// TwinCAT 3 PLC project NitroLogger
// Title: Tc_EventLogger
// Company: Reinova s.p.a.
// Author: Lorenzo Musco
// ProjectVersion: 1.1.2.6
// Description: This library wrap a Function block around the pre-existing TcLog in order to avoid cyclic call to the logger.
// ProgramVersion: 3.1.4024.0
// libraries:
//   Tc2_Standard, * (Beckhoff Automation GmbH)
//   Tc2_System, * (Beckhoff Automation GmbH)
//   Tc2_Utilities, * (Beckhoff Automation GmbH)
//   Tc3_Module, * (Beckhoff Automation GmbH)
//   TcLog, * (Benedikt Geisler)
//   Base Interfaces,newest,System
//   Tc3_DynamicMemory,1.0.2.0,Beckhoff Automation GmbH
// project tree:
//   / PlcTask.TcTTO
//   POUs/FB/ FB_EventLogger.TcPOU, FB_EventLoggerCore.TcPOU, FB_LogTrig.TcPOU, LogLevelToAdsLogMsgType.TcPOU
//   POUs/StringBuilder/ StringBuilder.TcPOU
//   POUs/StringBuilder/_Interfaces/ ILimitedStringBuilder.TcIO, IStringBuilder.TcIO
//   POUs/Utils/ AnyToString.TcPOU, DateTime.TcPOU, DeleteOldFiles.TcPOU, DynamicStringBuffer.TcPOU, GetFileAgeInSeconds.TcPOU
//   POUs/Utils/_DataTypes/ DeleteFilesState.TcDUT, PersistToFileState.TcDUT
//   POUs/_DataTypes/ Error.TcDUT, ErrorCodes.TcDUT, LoggingConfiguration.TcDUT, LogLevels.TcDUT, RollingIntervals.TcDUT
//   Version/ Global_Version.TcGVL
// real-time tasks:
//   TASK PlcTask: cycle T#10ms, priority 20, ADS port 350

CONFIGURATION NitroLogger
    RESOURCE PLC ON TwinCAT3
        TASK PlcTask(INTERVAL := T#10ms, PRIORITY := 20);
        PROGRAM MAIN WITH PlcTask : MAIN;
    END_RESOURCE
END_CONFIGURATION

// ---- POUs/Utils/_DataTypes/DeleteFilesState.TcDUT
// States for state machine used in `DeleteOldFiles`.
{attribute 'qualified_only'}
{attribute 'strict'}
TYPE INTERNAL DeleteFilesState :
(
	Idle := 0,
  SearchNextFile,
  WaitUntilExecutionDone,
  ProcessFoundFiles,
  CheckIfFileIsDirectory,
  CheckFileTime,
  DeleteFile,
  FileDeleted
);
END_TYPE

// ---- POUs/Utils/_DataTypes/PersistToFileState.TcDUT
// States for state machine used in `DynamicStringBuffer.PersistToFile`
{attribute 'qualified_only'}
{attribute 'strict'}
TYPE INTERNAL PersistToFileState :
(
	Idle := 0,
  OpenFile,
  GetStringFromFifo,
  AppendDataToFile,
  CloseFile
);
END_TYPE

// ---- POUs/_DataTypes/Error.TcDUT
/// This is the error type used in this library.
TYPE Error :
STRUCT
  /// `TRUE` signals an active error
	Active : BOOL;
  /// Error code of type `ErrorCodes`
	Code : INT;
  /// Plain text error message
	Info : Tc2_System.T_MaxString;
END_STRUCT
END_TYPE

// ---- POUs/_DataTypes/ErrorCodes.TcDUT
/// Provides error codes for TcLogCore
{attribute 'qualified_only'}
{attribute 'strict'}
{attribute 'to_string'}
TYPE ErrorCodes : 
(
	None := 0,
	OpeningFileFailed,
	WritingToFileFailed,
	ClosingFileFailed,
	EnumeratingFilesInSpecifiedDirectoryFailed,
	DeletingFileFailed,
	FifoOverflow
);
END_TYPE

// ---- POUs/_DataTypes/LoggingConfiguration.TcDUT
/// Configuration of TcLogCore
TYPE LoggingConfiguration :
STRUCT
  /// File name where the logs should be written to. Should not include path.
	FileName : Tc2_System.T_MaxString;
  /// File path where the logs should be written to. Will be prefixed to `FileName`
	FilePath : Tc2_System.T_MaxString;
  /// Whether to include the instance path of TcLog into the log message or not.
	IncludeInstancePath : BOOL;
  /// Whether to write the logs to ADS output or not.
	WriteToAds : BOOL;
  /// Rolling interval: when to create a new log file.
	RollingInterval : RollingIntervals;
  /// What is the minimum log level that gets logged?
	MinimumLevel : LogLevels;
  /// Which delimiter should be used between the different parts of the log string?
	Delimiter : STRING(1);
  /// When should old log files be deleted? Unit: days. Set it to `0` if log files should never be deleted. 
	LogFileLifespan : UINT;
  /// Format of timestamp. See `TcLogCore.TimestampFormat` for formatting options.
	TimestampFormat : STRING;
END_STRUCT
END_TYPE

// ---- POUs/_DataTypes/LogLevels.TcDUT
/// Log level of message to be logged.
{attribute 'qualified_only'}
{attribute 'strict'}
{attribute 'to_string'}
TYPE LogLevels :
(
	Debug := 0,
	Information,
	Warning,
	Error,
	Fatal
);
END_TYPE

// ---- POUs/_DataTypes/RollingIntervals.TcDUT
/// Rolling interval to create a new log file when expired. 
{attribute 'qualified_only'}
{attribute 'strict'}
{attrivute 'to_string'}
TYPE RollingIntervals :
(
	None := 0,
	Hourly,
	Daily,
	Monthly
);
END_TYPE

// ---- Version/Global_Version.TcGVL
{attribute 'TcGenerated'}
{attribute 'no-analysis'}
{attribute 'linkalways'}
// This function has been automatically generated from the project information.
VAR_GLOBAL CONSTANT
	{attribute 'const_non_replaced'}
	stLibVersion_Tc_EventLogger : ST_LibVersion := (iMajor := 1, iMinor := 1, iBuild := 2, iRevision := 6, nFlags := 1, sVersion := '1.1.2.6');
END_VAR

// ---- POUs/StringBuilder/_Interfaces/ILimitedStringBuilder.TcIO
{attribute 'hide'}
INTERFACE INTERNAL ILimitedStringBuilder

METHOD Append : IStringBuilder // Append text TO t current build STRING.
VAR_INPUT
    Text : Tc2_System.T_MaxString; //Text to append to current build string
END_VAR
END_METHOD

METHOD AppendIf : IStringBuilder
VAR_INPUT
    Condition : BOOL;
    Text : Tc2_System.T_MaxString;
END_VAR
END_METHOD

METHOD Reset : ILimitedStringBuilder //Reset current build STRING TO an empty STRING.
END_METHOD

METHOD ToString : Tc2_System.T_MaxString //Returns current build STRING.
END_METHOD

END_INTERFACE

// ---- POUs/StringBuilder/_Interfaces/IStringBuilder.TcIO
{attribute 'hide'}
INTERFACE INTERNAL IStringBuilder

METHOD Append : IStringBuilder // Append text TO t current build STRING.
VAR_INPUT
    Text : Tc2_System.T_MaxString; //Text to append to current build string
END_VAR
END_METHOD

METHOD AppendIf : IStringBuilder
VAR_INPUT
    Condition : BOOL;
    Text : Tc2_System.T_MaxString;
END_VAR
END_METHOD

METHOD InsertAtLocation : IStringBuilder
VAR_INPUT
    Text : Tc2_System.T_MaxString;
    Position : INT;
END_VAR
END_METHOD

METHOD PadLeft : IStringBuilder
VAR_INPUT
    Text : Tc2_System.T_MaxString; // Text to append to current build string
    Length : INT; // Total length of text + padding
    Char : STRING(1); // Character to be padded left of text
END_VAR
END_METHOD

METHOD Reset : ILimitedStringBuilder //Reset current build STRING TO an empty STRING.
END_METHOD

METHOD ToString : Tc2_System.T_MaxString //Returns current build STRING.
END_METHOD

END_INTERFACE

// ---- POUs/FB/FB_EventLogger.TcPOU
{attribute 'reflection'} 
FUNCTION_BLOCK FB_EventLogger EXTENDS TcLog
VAR
	_WorkString			: Tc2_System.T_MaxString;
	isSpammable			: BOOL;
	
	OldsCompletedString, NewCompletedString : T_MaxString;
END_VAR

METHOD Append : REFERENCE TO FB_EventLogger
VAR_INPUT
	sString		: T_MaxString;
END_VAR

VAR_INST
	OldString 	: T_MaxString;
END_VAR
_WorkString := CONCAT(_WorkString, sString);

Append REF= THIS^;
END_METHOD

METHOD CanSpam : REFERENCE TO FB_EventLogger
VAR
	
END_VAR
isSpammable := TRUE; 
CanSpam REF= THIS^;
END_METHOD

/// Logs the log string in DEBUG level.
METHOD Debug : BOOL
VAR_INPUT
  	message : T_MaxString; 
END_VAR
_WorkString := CONCAT(_WorkString, message);
NewCompletedString := _WorkString;
_WorkString := '';

IF NewCompletedString <> OldsCompletedString OR isSpammable THEN
	SUPER^.Debug(NewCompletedString);
	OldsCompletedString := NewCompletedString;
	isSpammable := FALSE;
END_IF
END_METHOD

/// Logs the log string in ERROR level.
METHOD Error : BOOL
VAR_INPUT
  	message : T_MaxString; 
END_VAR
_WorkString := CONCAT(_WorkString, message);
NewCompletedString := _WorkString;
_WorkString := '';

IF NewCompletedString <> OldsCompletedString THEN
	SUPER^.Error(NewCompletedString);
	OldsCompletedString := NewCompletedString;
	isSpammable := FALSE;
END_IF
END_METHOD

/// Logs the log string in FATAL level.
METHOD Fatal : BOOL
VAR_INPUT
  	message : T_MaxString; 
END_VAR
_WorkString := CONCAT(_WorkString, message);
NewCompletedString := _WorkString;
_WorkString := '';

IF NewCompletedString <> OldsCompletedString THEN
	SUPER^.Error(NewCompletedString);
	OldsCompletedString := NewCompletedString;
	isSpammable := FALSE;
END_IF
END_METHOD

/// Logs the log string in INFORMATION level.
METHOD Information : BOOL
VAR_INPUT
  	message : T_MaxString; 
END_VAR
_WorkString := CONCAT(_WorkString, message);
NewCompletedString := _WorkString;
_WorkString := '';

IF NewCompletedString <> OldsCompletedString THEN
	SUPER^.Information(NewCompletedString);
	OldsCompletedString := NewCompletedString;
	isSpammable := FALSE;
END_IF
END_METHOD

/// Initializes the reference to the core logger. Should only be called once from the core logger directly.
METHOD PUBLIC Init : BOOL
VAR_INPUT
  /// Reference to TcLoggerCore instance.
  ref2Core : ILogCore; 
END_VAR
SUPER^.Init(ref2Core);
END_METHOD

/// Logs the log string in WARNING level.
METHOD Warning : BOOL
VAR_INPUT
  	message : T_MaxString; 
END_VAR
_WorkString := CONCAT(_WorkString, message);
NewCompletedString := _WorkString;
_WorkString := '';

IF NewCompletedString <> OldsCompletedString THEN
	SUPER^.Warning(NewCompletedString);
	OldsCompletedString := NewCompletedString;
	isSpammable := FALSE;
END_IF
END_METHOD

END_FUNCTION_BLOCK

// ---- POUs/FB/FB_EventLoggerCore.TcPOU
FUNCTION_BLOCK FB_EventLoggerCore EXTENDS TcLogCore
VAR_INPUT
END_VAR
VAR_OUTPUT
END_VAR
VAR
END_VAR

END_FUNCTION_BLOCK

// ---- POUs/FB/FB_LogTrig.TcPOU
/// This function block can be used to log on rising or falling edges.
/// For each signal that should be watched, a separate instance of `TcLogTrig` 
/// must be created.
FUNCTION_BLOCK FB_LogTrig EXTENDS TcLog

/// Logs data on falling edge of `CLK`.
{attribute 'hide_all_locals'}
METHOD OnFallingEdge : REFERENCE TO TcLog
VAR_INPUT
  /// Falling edge triggers logging the data.
  CLK : BOOL; 
END_VAR
VAR_INST
    fTrig : Tc2_Standard.F_TRIG;
END_VAR
fTrig(CLK:=CLK);

SUPER^.OnCondition(fTrig.Q);

OnFallingEdge REF= THIS^;
END_METHOD

/// Logs data on rising edge of `CLK`.
{attribute 'hide_all_locals'}
METHOD OnRisingEdge : REFERENCE TO TcLog
VAR_INPUT
  /// Rising edge logs data.
  CLK : BOOL; 
END_VAR
VAR_INST
    rTrig : Tc2_Standard.R_TRIG;
END_VAR
rTrig(CLK:=CLK);

SUPER^.OnCondition(rTrig.Q);

OnRisingEdge REF= THIS^;
END_METHOD

END_FUNCTION_BLOCK

// ---- POUs/FB/LogLevelToAdsLogMsgType.TcPOU
// Converts TcLog.LogLevels into Tc2_System.ADSLOG_MSGTYPEs.
{attribute 'hide'}
FUNCTION INTERNAL LogLevelToAdsLogMsgType : DWORD
VAR_INPUT
  logLevel : LogLevels;
END_VAR
VAR
  _retVal : DWORD;
END_VAR

CASE logLevel OF
  LogLevels.Debug, LogLevels.Information:
    _retVal := Tc2_System.ADSLOG_MSGTYPE_HINT;
  LogLevels.Warning:
    _retVal := Tc2_System.ADSLOG_MSGTYPE_WARN;
  LogLevels.Error, LogLevels.Fatal:
    _retVal := Tc2_System.ADSLOG_MSGTYPE_ERROR;
  ELSE
    _retVal := Tc2_System.ADSLOG_MSGTYPE_HINT;
END_CASE

LogLevelToAdsLogMsgType := _retVal;

END_FUNCTION

// ---- POUs/StringBuilder/StringBuilder.TcPOU
FUNCTION_BLOCK INTERNAL StringBuilder IMPLEMENTS IStringBuilder, ILimitedStringBuilder
VAR
  {attribute 'hide'}
  _workString : Tc2_System.T_MaxString;
END_VAR

METHOD PUBLIC Append : IStringBuilder // Append text TO t current build STRING.
VAR_INPUT
  text : Tc2_System.T_MaxString; //text to append to current build string
END_VAR
_workString:= Tc2_Standard.CONCAT(_workString,text);
Append := THIS^;
END_METHOD

METHOD PUBLIC AppendIf : IStringBuilder
VAR_INPUT
  condition : BOOL;
  text : Tc2_System.T_MaxString;
END_VAR
IF condition THEN
  _workString:= Tc2_Standard.CONCAT(_workString,text);
END_IF
AppendIf := THIS^;
END_METHOD

METHOD PUBLIC InsertAtLocation : IStringBuilder
VAR_INPUT
  text : Tc2_System.T_MaxString;
  position : INT;
END_VAR
_workString := Tc2_Standard.INSERT(_workSTring,text,position);
InsertAtLocation  := THIS^;
END_METHOD

METHOD PadLeft : IStringBuilder
VAR_INPUT
  text : Tc2_System.T_MaxString; // Text to append to current build string
  length : INT; // Total length of text + padding
  char : STRING(1); // Character to be padded left of text
END_VAR
VAR
  i : INT;
  padLength : INT;
END_VAR
// Add left padding
padLength := Tc2_Standard.LEN(text) - length;
FOR i := 1 TO padLength DO
  _workString:= Tc2_Standard.CONCAT(_workString, char);
END_FOR

// Add text
_workString:= Tc2_Standard.CONCAT(_workString,text);

PadLeft := THIS^;
END_METHOD

METHOD PUBLIC Reset : ILimitedStringBuilder //Reset current build STRING TO an empty STRING.
_workString:='';
Reset := THIS^;
END_METHOD

METHOD PUBLIC ToString : Tc2_System.T_MaxString //Returns current build STRING.
ToString := _workString;
END_METHOD

END_FUNCTION_BLOCK

// ---- POUs/Utils/AnyToString.TcPOU
/// Converts value of input data to string, where the input type can be any of 
/// the standard data types.
FUNCTION AnyToString : Tc2_System.T_MaxString
VAR_INPUT
  /// Input data
  data : ANY;
END_VAR
VAR
  _anyByte : POINTER TO BYTE;
  _anyUSINT : POINTER TO USINT;
  _anyInt : POINTER TO INT;
  _anyUInt : POINTER TO UINT;
  _anyUDInt : POINTER TO UDINT;
  _anySInt : POINTER TO SINT;
  _anyDInt : POINTER TO DINT;
  _anyLInt : POINTER TO LINT;
  _anyULInt : POINTER TO ULINT;
  _anyWord : POINTER TO WORD;
  _anyLWord : POINTER TO LWORD;
  _anyReal : POINTER TO REAL;
  _anyLReal : POINTER TO LREAL;
  _anyDateAndTime : POINTER TO DATE_AND_TIME;
  _anyDate : POINTER TO DATE;
  _anyTime : POINTER TO TIME;
  _anyWString : POINTER TO WSTRING;
  _anyTOD : POINTER TO TOD;
  _anyString : POINTER TO STRING;
  _string : T_MAXSTRING;
  _wString : WSTRING;
END_VAR

IF data.TypeClass = __SYSTEM.TYPE_CLASS.TYPE_BYTE THEN
  _anyByte := data.pValue;
  AnyToString := BYTE_TO_STRING(_anyByte^);
    
ELSIF data.TypeClass = __SYSTEM.TYPE_CLASS.TYPE_INT THEN
  _anyInt := data.pValue;
  AnyToString := INT_TO_STRING(_anyInt^);
    
ELSIF data.TypeClass = __SYSTEM.TYPE_CLASS.TYPE_UINT THEN
  _anyUInt := data.pValue;
  AnyToString := UINT_TO_STRING(_anyUInt^);
    
ELSIF data.TypeClass = __SYSTEM.TYPE_CLASS.TYPE_UDINT THEN
  _anyUDInt := data.pValue;
  AnyToString := UDINT_TO_STRING(_anyUDInt^);
    
ELSIF data.TypeClass = __SYSTEM.TYPE_CLASS.TYPE_SINT THEN
  _anySInt := data.pValue;
  AnyToString := SINT_TO_STRING(_anySInt^);
    
ELSIF data.TypeClass = __SYSTEM.TYPE_CLASS.TYPE_USINT THEN
  _anyUSInt := data.pValue;
  AnyToString := USINT_TO_STRING(_anyUSInt^);
    
ELSIF data.TypeClass = __SYSTEM.TYPE_CLASS.TYPE_DINT THEN
  _anyDInt := data.pValue;
  AnyToString := DINT_TO_STRING(_anyDInt^);
    
ELSIF data.TypeClass = __SYSTEM.TYPE_CLASS.TYPE_LINT THEN
  _anyLInt := data.pValue;
  AnyToString := LINT_TO_STRING(_anyLInt^);
      
ELSIF data.TypeClass = __SYSTEM.TYPE_CLASS.TYPE_ULINT THEN
  _anyULInt := data.pValue;
  AnyToString := ULINT_TO_STRING(_anyULInt^);
  
ELSIF data.TypeClass = __SYSTEM.TYPE_CLASS.TYPE_WORD THEN
  _anyWord := data.pValue;
  AnyToString := WORD_TO_STRING(_anyWord^);
    
ELSIF data.TypeClass = __SYSTEM.TYPE_CLASS.TYPE_LWORD THEN
  _anyLWord := data.pValue;
  AnyToString := LWORD_TO_STRING(_anyLWord^);
  
ELSIF data.TypeClass = __SYSTEM.TYPE_CLASS.TYPE_REAL THEN
  _anyReal := data.pValue;
  AnyToString := REAL_TO_STRING(_anyReal^);
  
ELSIF data.TypeClass = __SYSTEM.TYPE_CLASS.TYPE_LREAL THEN
  _anyLReal := data.pValue;
  AnyToString := LREAL_TO_STRING(_anyLReal^);
  
ELSIF data.TypeClass = __SYSTEM.TYPE_CLASS.TYPE_DATEANDTIME THEN
  _anyDateAndTime := data.pValue;
  AnyToString := DT_TO_STRING(_anyDateAndTime^);  
  
ELSIF data.TypeClass = __SYSTEM.TYPE_CLASS.TYPE_DATE THEN
  _anyDate := data.pValue;
  AnyToString := DATE_TO_STRING(_anyDate^);
  
ELSIF data.TypeClass = __SYSTEM.TYPE_CLASS.TYPE_TIME THEN
  _anyTime := data.pValue;
  AnyToString := TIME_TO_STRING(_anyTime^);
  
ELSIF data.TypeClass = __SYSTEM.TYPE_CLASS.TYPE_STRING THEN
  _anyString := data.pValue;
  AnyToString := _anyString^;
  
ELSIF data.TypeClass = __SYSTEM.TYPE_CLASS.TYPE_WSTRING THEN
  _anyWString := data.pValue;
  _wString := _anyWString^;
  Tc2_Utilities.WSTRING_TO_STRING2(ADR(_string), ADR(_wString), SIZEOF(_wString));
  AnyToString := _string;
  
ELSIF data.TypeClass = __SYSTEM.TYPE_CLASS.TYPE_TIMEOFDAY THEN
  _anyTOD := data.pValue;
  AnyToString := TOD_TO_STRING(_anyTOD^);
  
ELSE
  AnyToString := TO_STRING(data.pValue^);
END_IF

END_FUNCTION

// ---- POUs/Utils/DateTime.TcPOU
/// Generate time data in different formats.
{attribute: 'hide_all_locals'}
FUNCTION_BLOCK DateTime
VAR
  _localSystemTime : Tc2_Utilities.FB_LocalSystemTime;
  _getSystemTime : Tc2_System.GETSYSTEMTIME;
  _timeZoneInfo : Tc2_Utilities.FB_GetTimeZoneInformation;
  _localTime : Tc2_Utilities.FB_SystemTimeToTzSpecificLocalTime;
  _localSystemTimeValid : Tc2_Standard.R_TRIG;
  _utcTime : Tc2_Utilities.FB_TzSpecificLocalTimeToFileTime;
END_VAR

// Get local system time
_localSystemTime(
  sNetID  :=  '',
  bEnable :=  TRUE,
  dwCycle :=  1,
  dwOpt :=  1,
  tTimeout:=  DEFAULT_ADS_TIMEOUT
);

// Get timezone information
_timeZoneInfo(
  sNetID := '',
  bExecute := TRUE,
  tTimeout := DEFAULT_ADS_TIMEOUT);

// Convert local time to utc time
_utcTime(
  in := THIS^.AsLocalFileTime,
  tzInfo := _timeZoneInfo.tzInfo);
  
// Finished retrieving time data
_localSystemTimeValid(CLK := _localSystemTime.bValid);

/// Returns local time as `Tc2_Utilities.T_FILETIME`.
{attribute 'monitoring':='variable'}
PROPERTY AsLocalFileTime : Tc2_Utilities.T_FILETIME
GET
AsLocalFileTime := SYSTEMTIME_TO_FILETIME(THIS^.AsLocalSystemTime);
END_GET
END_PROPERTY

/// Returns local time as `Tc2_Utilities.TIMESTRUCT`.
{attribute 'monitoring':='variable'}
PROPERTY AsLocalSystemTime : Tc2_Utilities.TIMESTRUCT
GET
AsLocalSystemTime := _localSystemTime.systemTime;
END_GET
END_PROPERTY

/// Returns local time as string.
{attribute 'monitoring':='variable'}
PROPERTY AsLocalSystemTimeString : Tc2_System.T_MAXSTRING
GET
AsLocalSystemTimeString := Tc2_Utilities.SYSTEMTIME_TO_STRING(THIS^.AsLocalSystemTime);
END_GET
END_PROPERTY

/// Returns UTC time as `Tc2_Utilities.T_FILETIME`.
{attribute 'monitoring':='variable'}
PROPERTY AsUtcFileTime : Tc2_Utilities.T_FILETIME
GET
AsUtcFileTime := _utcTime.out;
END_GET
END_PROPERTY

/// When calling `DateTime` the first time, it takes some time until all time and timezone information is available.
/// `Done` is `TRUE` for one cycle, once all the data is ready. 
{attribute 'monitoring':='call'}
PROPERTY Done : BOOL
GET
Done := _localSystemTimeValid.Q;
END_GET
END_PROPERTY

// Replaces placeholders in format string by the actual time values.
{attribute 'hide_all_locals'}
{attribute 'hide'}
METHOD PRIVATE ReplaceFormatPlaceholder : STRING
VAR_INPUT
  format : STRING;
  length : INT;
  timeType : STRING(1);
END_VAR
VAR_INST
  i : INT;
  replaceString : STRING;
  timeString : STRING;
END_VAR
VAR
  localSystemTime : Tc2_Utilities.TIMESTRUCT;
END_VAR
localSystemTime := THIS^.AsLocalSystemTime;

IF    timeType = 'Y'  THEN timeString := TO_STRING(localSystemTime.wYear); 
ELSIF timeType = 'M'  THEN timeString := TO_STRING(localSystemTime.wMonth); 
ELSIF timeType = 'D'  THEN timeString := TO_STRING(localSystemTime.wDay); 
ELSIF timeType = 'h'  THEN timeString := TO_STRING(localSystemTime.wHour); 
ELSIF timeType = 'm'  THEN timeString := TO_STRING(localSystemTime.wMinute); 
ELSIF timeType = 's'  THEN timeString := TO_STRING(localSystemTime.wSecond); 
ELSIF timeType = 'i'  THEN timeString := TO_STRING(localSystemTime.wMilliseconds); 
ELSE
  timeString:='';
END_IF

replaceString := '';

IF length > Tc2_Standard.LEN(timeString) THEN
  FOR i:=1 TO length - Tc2_Standard.LEN(timeString) DO
    replaceString := Tc2_Standard.CONCAT(replaceString, '0');
  END_FOR
  replaceString := Tc2_Standard.CONCAT(replaceString, timeString);
ELSE
  replaceString := Tc2_Standard.RIGHT(timeString, length);
END_IF

ReplaceFormatPlaceholder := Tc2_Standard.REPLACE(format, replaceString, length, Tc2_Standard.FIND(format, timeType));
END_METHOD

/// Returns a formatted string containing the actual time information 
/// - `Y` : year
/// - `M` : month
/// - `D` : day
/// - `h` : hour 
/// - `m` : minute
/// - `s` : second
/// - `i` : millisecond
/// 
/// Example:    
/// _YYMMDD-hh:mm:ss:iii_   
/// => _20210812-12:30:22:123_
{attribute 'hide_all_locals'}
METHOD ToFormatString : Tc2_System.T_MaxString
VAR_INPUT
  /// Format the timestamp should have.
  format : STRING;
END_VAR
VAR_INST
  inputString : STRING;
  char : STRING(1);
  formattedString : Tc2_System.T_MaxString;
END_VAR
VAR
  year : INT := 0;
  month : INT := 0;
  day : INT := 0;
  hour : INT := 0;
  minute : INT := 0;
  second : INT := 0;
  millisecond : INT := 0;
END_VAR
VAR CONSTANT
  ValidFormat : STRING := 'YMDhms';
END_VAR
// Parses "format" and returns a adequatly formatted string containing the time information
inputString := format;

WHILE Tc2_Standard.LEN(inputString) > 0 DO
  char := Tc2_Standard.LEFT(inputString, 1);
  
  IF    char = 'Y' THEN   year := year + 1;
  ELSIF char = 'M' THEN month := month + 1;
  ELSIF char = 'D' THEN day := day + 1;
  ELSIF char = 'h' THEN hour := hour + 1;
  ELSIF char = 'm' THEN minute := minute + 1;
  ELSIF char = 's' THEN   second := second + 1;
  ELSIF char = 'i' THEN   millisecond := millisecond + 1;
  END_IF
  
  inputString := Tc2_Standard.DELETE(inputString, 1, 1);
END_WHILE

formattedString := ReplaceFormatPlaceholder(format, year, 'Y');
formattedString := ReplaceFormatPlaceholder(formattedString, month, 'M');
formattedString := ReplaceFormatPlaceholder(formattedString, day, 'D');
formattedString := ReplaceFormatPlaceholder(formattedString, hour, 'h');
formattedString := ReplaceFormatPlaceholder(formattedString, minute, 'm');
formattedString := ReplaceFormatPlaceholder(formattedString, second, 's');
formattedString := ReplaceFormatPlaceholder(formattedString, millisecond, 'i');

ToFormatString := formattedString;
END_METHOD

END_FUNCTION_BLOCK

// ---- POUs/Utils/DeleteOldFiles.TcPOU
{attribute 'hide_all_locals'}
FUNCTION_BLOCK INTERNAL DeleteOldFiles
VAR_INPUT
  StartScan : BOOL; // Rising edge starts scan for out-of-date log files and deletes them.
  ExpirationInDays : UINT; // Files will be deleted if older than n days
  FilePath : Tc2_System.T_MaxString; // Path to files to be deleted
  FileName : Tc2_System.T_MaxString; // Only files which match this filename will be deleted
  CurrentUtcTime : Tc2_Utilities.T_FILETIME; // Current time  as UTC
END_VAR
VAR_OUTPUT
  Error : Error; // Error information
END_VAR
VAR CONSTANT
  OneDayInSeconds : LREAL := 24*3600.0;
  MaxNumberOfFiles : UDINT := 100;
END_VAR
VAR
  _state : DeleteFilesState := DeleteFilesState.Idle;
  
  _enumFindFileList : Tc2_Utilities.FB_EnumFindFileList;
  _enumBusy : Tc2_Standard.F_TRIG;
  _fileDelete : Tc2_System.FB_FileDelete;
  _fileDeleteBusy : Tc2_Standard.F_TRIG;
  _listOfFiles : ARRAY[1..100] OF Tc2_Utilities.ST_FindFileEntry;
  _deleteFileIndex : UDINT;
  _fileNameToDelete : Tc2_System.T_MaxString;
  _commandType : Tc2_Utilities.E_EnumCmdType;
  _fileDeleted : BOOL;
  _startFileDelete: BOOL;
END_VAR

// State machine to delete all due files.
// It first enumerates all files in the specified directory
// and then deletes all files that have overpassed the specified due date
_startFileDelete := FALSE;

CASE _state OF
  DeleteFilesState.Idle:
    IF StartScan THEN
      _commandType:= eEnumCmd_First;
      _deleteFileIndex := 1;
      _state := DeleteFilesState.SearchNextFile;
    END_IF
    
  DeleteFilesState.SearchNextFile:
    IF _enumBusy.Q THEN
      _state := DeleteFilesState.WaitUntilExecutionDone;
    END_IF
    
  DeleteFilesState.WaitUntilExecutionDone:
    IF NOT _enumFindFileList.bError THEN
      IF NOT _enumFindFileList.bEOE THEN
        IF _enumFindFileList.nFindFiles < MaxNumberOfFiles THEN
          _state := DeleteFilesState.SearchNextFile;
        ELSE
          _commandType := eEnumCmd_Abort;
          _state := DeleteFilesState.ProcessFoundFiles;
        END_IF
      ELSE
        _state := DeleteFilesState.ProcessFoundFiles;
      END_IF
    ELSE
      _state := DeleteFilesState.Idle;
    END_IF
    
  DeleteFilesState.ProcessFoundFiles:
    IF _deleteFileIndex > _enumFindFileList.nFindFiles THEN
      _state := DeleteFilesState.Idle;
    ELSE
      _state := DeleteFilesState.CheckIfFileIsDirectory;
    END_IF
    
  DeleteFilesState.CheckIfFileIsDirectory:
    IF NOT _listOfFiles[_deleteFileIndex].fileAttributes.bDirectory THEN
      _state := DeleteFilesState.CheckFileTime;
    ELSE
      _deleteFileIndex := _deleteFileIndex + 1;
      _state := DeleteFilesState.ProcessFoundFiles;
    END_IF
    
  DeleteFilesState.CheckFileTime:   
    IF GetFileAgeInSeconds(CurrentUtcTime, _listOfFiles[_deleteFileIndex]) > (ExpirationInDays * OneDayInSeconds) THEN
      _state := DeleteFilesState.DeleteFile;
    ELSE
      _deleteFileIndex := _deleteFileIndex + 1;
      _state := DeleteFilesState.ProcessFoundFiles;
    END_IF
  
  DeleteFilesState.DeleteFile:
    _fileNameToDelete := Tc2_Standard.CONCAT(FilePath, _listOfFiles[_deleteFileIndex].sFileName);
    _startFileDelete := TRUE;
    
    IF _fileDeleteBusy.Q THEN
      _deleteFileIndex := _deleteFileIndex + 1;
      _fileDeleted := TRUE;
      _state := DeleteFilesState.FileDeleted;
    END_IF
    IF _fileDelete.bError THEN
      _state := DeleteFilesState.Idle;
    END_IF
    
  DeleteFilesState.FileDeleted:   
    // This state is needed to generate a rising edge for FB_FileDelete
    IF NOT _fileDeleted THEN
      _state := DeleteFilesState.ProcessFoundFiles;
    END_IF
    _fileDeleted := FALSE;

END_CASE

// Function blocks used in state machine

// Search files in given directory
_enumFindFileList(sNetId := '',
       eCmd := _commandType,
       sPathName := Tc2_Standard.CONCAT(FilePath, Tc2_Standard.CONCAT('*', FileName)),
       bExecute := (_state = DeleteFilesState.SearchNextFile) OR (_commandType = eEnumCmd_Abort AND _state <> DeleteFilesState.Idle),
       pFindList := ADR(_listOfFiles),
       cbFindList := SIZEOF(_listOfFiles),
       tTimeout := T#10S);
       
_enumBusy(CLK:=_enumFindFileList.bBusy);

// Delete files
_fileDelete(sNetId := '',
             sPathName := _fileNameToDelete,
             bExecute := _startFileDelete,
             tTimeout := T#10S);

_fileDeleteBusy(CLK := _fileDelete.bBusy);

// Error handling
Error.Active := FALSE;
Error.Code := ErrorCodes.None;
Error.Info := '';

IF _enumFindFileList.bError THEN
  Error.Active := TRUE;
  Error.Code := ErrorCodes.EnumeratingFilesInSpecifiedDirectoryFailed;
  Error.Info := Tc2_Standard.CONCAT('Enumerating files in specified directory failed. Error thrown by FB_EnumFindFileList. Consult Beckhoff InfoSys. Internal Error: ', UDINT_TO_STRING(_enumFindFileList.nErrId));
END_IF
      
IF _fileDelete.bError THEN
  Error.Active := TRUE;
  Error.Code := ErrorCodes.DeletingFileFailed;
  Error.Info := Tc2_Standard.CONCAT('Deleting expired log file in specified directory failed. Error thrown by FB_FileDelete. Consult Beckhoff InfoSys. Internal Error: ', UDINT_TO_STRING(_fileDelete.nErrId));
END_IF

END_FUNCTION_BLOCK

// ---- POUs/Utils/GetFileAgeInSeconds.TcPOU
{attribute 'hide'}
FUNCTION INTERNAL GetFileAgeInSeconds : DINT
VAR_INPUT
  currentUtcTime : Tc2_Utilities.T_FILETIME;
  findFileEntry : Tc2_Utilities.ST_FindFileEntry;
END_VAR
VAR
  _timeLastWriteAccess : Tc2_Utilities.T_ULARGE_INTEGER;
  _fileTimeAsULINT : Tc2_Utilities.T_ULARGE_INTEGER;
  _fileTimeDifference : Tc2_Utilities.T_ULARGE_INTEGER;
END_VAR
VAR CONSTANT
  OneSecondInOneHundredNanoSecondsIntervals : LREAL := 1000*1000*10;
END_VAR

// Local file time
_fileTimeAsULINT.dwLowPart := currentUtcTime.dwLowDateTime;
_fileTimeAsULINT.dwHighPart := currentUtcTime.dwHighDateTime;

// Write access is UTC
_timeLastWriteAccess.dwLowPart := findFileEntry.lastWriteTime.dwLowDateTime;
_timeLastWriteAccess.dwHighPart := findFileEntry.lastWriteTime.dwHighDateTime;
_fileTimeDifference := UInt64Sub64(_fileTimeAsULINT, _timeLastWriteAccess);

GetFileAgeInSeconds := LREAL_TO_DINT(UINT64_TO_LREAL(_fileTimeDifference)/(OneSecondInOneHundredNanoSecondsIntervals));

END_FUNCTION

// ---- POUs/Utils/DynamicStringBuffer.TcPOU
{attribute 'hide_all_locals'}
FUNCTION_BLOCK INTERNAL DynamicStringBuffer
VAR_OUTPUT
  Error : Error; // Error information of this FB
END_VAR
VAR
  _fifo : Tc2_Utilities.FB_StringRingBuffer; // Necessary to buffer log data until it has been written to file.
  _memoryManager : Tc3_DynamicMemory.FB_DynMem_Manager; // Memory manager, required by DynMem_Buffer.
  _dynamicMemoryBuffer : Tc3_DynamicMemory.FB_DynMem_Buffer(ipMemMan := _memoryManager); // Provides dynamic buffer for Fifo. Is extended automatically if more than the
                                                                   // default buffer size is needed.                  
  _busy : BOOL; // Buffer is busy; typically with writing data to the file system.
END_VAR

METHOD AddLine : BOOL
VAR_INPUT
  text : Tc2_System.T_MaxString; // Text to be added to the buffer
END_VAR
ResizeFifoBufferIfNecessary();
_fifo.A_AddTail(putValue := Tc2_Standard.CONCAT(Tc2_Standard.LEFT(text, 254), '$N'));
END_METHOD

METHOD AddString : BOOL
VAR_INPUT
  text : Tc2_System.T_MaxString; // String to be added to the buffer
END_VAR
ResizeFifoBufferIfNecessary();
_fifo.A_AddTail(putValue := text);
END_METHOD

METHOD PRIVATE AllocateBuffer : BOOL // Allocates buffer FOR the fifo.
VAR_INPUT
  bufferSize : UDINT; // Initial buffer size in BYTEs for fifo buffer.
END_VAR
_dynamicMemoryBuffer.CreateBuffer(nSize:=bufferSize, bReset:=TRUE);
_fifo.pBuffer := _dynamicMemoryBuffer.pBuffer;
_fifo.cbBuffer := bufferSize;
END_METHOD

{attribute 'monitoring':='call'}
PROPERTY Busy : BOOL
GET
Busy := _busy;
END_GET
SET // PRIVATE
_busy := Busy;
END_SET
END_PROPERTY

METHOD FB_exit : BOOL
VAR_INPUT
  bInCopyCode : BOOL; // if TRUE, the exit method is called for exiting an instance that is copied afterwards (online change).
END_VAR
_dynamicMemoryBuffer.Clear();
END_METHOD

METHOD FlushCache : BOOL
_fifo.A_Reset();
END_METHOD

METHOD INTERNAL Init : BOOL
VAR_INPUT
  bufferSize : UDINT; // Initial buffer size in BYTEs for fifo buffer.
END_VAR
AllocateBuffer(bufferSize);
END_METHOD

{attribute 'hide_all_locals'}
METHOD PersistToFile : BOOL
VAR_INPUT
  enable: BOOL; // TRUE starts persistence mechanism
  fileName : Tc2_System.T_MaxString; // File name including its path
END_VAR
VAR_INST
  state : PersistToFileState;
  
  fileOpen : Tc2_System.FB_FileOpen;
  fileHandle : UINT;
  
  fileWrite : Tc2_System.FB_FileWrite;
  lockFileWriteToForceRisingEdge : BOOL; // filePuts can only be executed every other cycle
                                         // since it needs a rising edge to execute.
  fileClose : Tc2_System.FB_FileClose;
  
  buffer : ARRAY[0..CONSTANTS.BufferSize] OF BYTE;
  currentBufferPos : UDINT;
  fifoHeadString : Tc2_System.T_MaxString;
  fifoHeadLength : UDINT;
  fifoHeadBytes : ARRAY[0..Tc2_System.Tc2_System.MAX_STRING_LENGTH] OF BYTE;
  i : UINT;
END_VAR
VAR CONSTANT
  NetId : STRING := '';
  Timeout : TIME := DEFAULT_ADS_TIMEOUT;
  MaxLogsPerCycle : UINT := DINT_TO_UINT(CONSTANTS.BufferSize / UDINT_TO_DINT(Tc2_System.MAX_STRING_LENGTH));
  MaxBufferPosition : UDINT := (SIZEOF(buffer)-Tc2_System.MAX_STRING_LENGTH);
END_VAR
// State machine
// Using if-statements instead of case for performance reasons:
// Some states execute instantly and allow thus the next state 
// to start within the same plc cycle.

// *** I D L E ***
IF state = PersistToFileState.Idle THEN
  lockFileWriteToForceRisingEdge := FALSE;
  IF _fifo.nCount > 0 AND enable THEN 
    lockFileWriteToForceRisingEdge := FALSE;
    state := PersistToFileState.OpenFile;
  END_IF
END_IF
    
// *** O P E N   F I L E ***
fileOpen(sNetId := NetId, sPathName := fileName, nMode := FOPEN_MODEAPPEND OR FOPEN_MODETEXT, 
           ePath := PATH_GENERIC, bExecute := (state = PersistToFileState.OpenFile), tTimeout := Timeout,
           hFile => fileHandle);

IF state = PersistToFileState.OpenFile THEN
  IF fileOpen.bError THEN
    state := PersistToFileState.CloseFile;
  ELSIF NOT fileOpen.bBusy THEN
    state := PersistToFileState.GetStringFromFifo; 
  END_IF
END_IF 

// *** P O P   F R O M   F I F O ***
IF state = PersistToFileState.GetStringFromFifo THEN
  IF NOT lockFileWriteToForceRisingEdge THEN
    currentBufferPos := 0;
    FOR i:=0 TO MaxLogsPerCycle DO
      IF _fifo.nCount <= 0 THEN EXIT; END_IF
      IF currentBufferPos >= MaxBufferPosition THEN EXIT; END_IF
      
      _fifo.A_RemoveHead(getValue => fifoHeadString); 
      fifoHeadBytes := MAXSTRING_TO_BYTEARR(fifoHeadString);
      fifoHeadLength := INT_TO_UDINT(LEN(fifoHeadString));
      MEMCPY(
        destAddr  :=  ADR(buffer) + SIZEOF(BYTE) * currentBufferPos,
        srcAddr   :=  ADR(fifoHeadBytes),
        n     :=  fifoHeadLength);    
      currentBufferPos := currentBufferPos + fifoHeadLength;  
    END_FOR
    state := PersistToFileState.AppendDataToFile;
  END_IF
  lockFileWriteToForceRisingEdge := FALSE;
END_IF
  
// *** W R I T E   T O   F I L E ***
fileWrite(
  sNetId := NetId, 
  hFile := fileHandle, 
  pWriteBuff := ADR(buffer),
  cbWriteLen := currentBufferPos,
  bExecute := state = PersistToFileState.AppendDataToFile, 
  tTimeout := Timeout); 

IF state = PersistToFileState.AppendDataToFile THEN
  lockFileWriteToForceRisingEdge := TRUE;   
  IF fileWrite.bError THEN
    state := PersistToFileState.CloseFile;
  ELSIF _fifo.nCount > 0 AND NOT fileWrite.bBusy THEN
    state := PersistToFileState.GetStringFromFifo; 
  ELSIF _fifo.nCount = 0 THEN
    state := PersistToFileState.CloseFile;
  END_IF
END_IF
    
// *** C L O S E   F I L E ***
fileClose(
  sNetId := NetId, hFile := fileHandle, 
  bExecute := (state = PersistToFileState.CloseFile), tTimeout := Timeout);

IF state = PersistToFileState.CloseFile THEN
  IF NOT fileClose.bBusy THEN state := PersistToFileState.Idle; END_IF
END_IF

// Close file in case of error
IF fileOpen.bError THEN state := PersistToFileState.CloseFile; END_IF
IF fileWrite.bError THEN state := PersistToFileState.CloseFile; END_IF
IF NOT _fifo.bOk AND _fifo.nCount > 0 AND state <> PersistToFileState.Idle THEN 
  state := PersistToFileState.CloseFile; 
END_IF

// Error handling
IF fileOpen.bError THEN
  Error.Active := TRUE;
  Error.Code := ErrorCodes.OpeningFileFailed;
  Error.Info := Tc2_Standard.CONCAT('Opening file failed. Error thrown by FB_FileOpen. Consult Beckhoff InfoSys. Internal Error: ', UDINT_TO_STRING(fileOpen.nErrId));
ELSIF fileWrite.bError THEN
  Error.Active := TRUE;
  Error.Code := ErrorCodes.WritingToFileFailed;
  Error.Info := Tc2_Standard.CONCAT('Writing to file failed. Error thrown by FB_FileWrite. Consult Beckhoff InfoSys. Internal Error: ', UDINT_TO_STRING(fileWrite.nErrId));
ELSIF fileClose.bError THEN
  Error.Active := TRUE;
  Error.Code := ErrorCodes.ClosingFileFailed;
  Error.Info := Tc2_Standard.CONCAT('Closing file failed. Error thrown by FB_FileClose. Consult Beckhoff InfoSys. Internal Error: ', UDINT_TO_STRING(fileClose.nErrId));
ELSIF NOT _fifo.bOk AND _fifo.nCount > 0 THEN
  Error.Active := TRUE;
  Error.Code := ErrorCodes.FifoOverflow;
  Error.Info := 'FIFO overflow. Check if plc has enough free memory.';
ELSE
  Error.Active := FALSE;
  Error.Code := ErrorCodes.None;
  Error.Info := '';
END_IF

// Set busy state
Busy := (state <> PersistToFileState.Idle OR _fifo.nCount > 0);

(* Uncomment for cyclic logging of state machine, buffer usage & errors

ADSLOGSTR(ADSLOG_MSGTYPE_LOG, 
  Tc2_Standard.CONCAT('****DynamicStringBuffer.state:', 
  Tc2_Standard.CONCAT(UINT_TO_STRING(state),
  Tc2_Standard.CONCAT(', DynamicStringBuffer.hFile:', UINT_TO_STRING(hFile)))), '');

ADSLOGSTR(ADSLOG_MSGTYPE_LOG, 
  Tc2_Standard.CONCAT('****Fifo: used ', 
  Tc2_Standard.CONCAT(UDINT_TO_STRING(Fifo.cbSize),
  Tc2_Standard.CONCAT(' of ', UDINT_TO_STRING(Fifo.cbBuffer)))), '');
  
IF Error.Active THEN
  ADSLOGSTR(ADSLOG_MSGTYPE_LOG, 
    Tc2_Standard.CONCAT('****DynamicStringBuffer.Error: ', Error.Info), 
    '');  
END_IF
*)
END_METHOD

METHOD PopHead : Tc2_System.T_MaxString
VAR_INST
  headString : Tc2_System.T_MaxString;
END_VAR
_fifo.A_RemoveHead(getValue => headString);
PopHead := headString;
END_METHOD

// Resizes the buffer for the FIFO if necessary
METHOD PRIVATE ResizeFifoBufferIfNecessary : BOOL
VAR
  requiredSize : UDINT;
  newSize : DINT;
END_VAR
requiredSize := _fifo.cbSize + (Tc2_System.Tc2_System.MAX_STRING_LENGTH + INT_TO_UDINT(Constants.FifoOverhead));

IF requiredSize > _fifo.cbBuffer THEN
  _dynamicMemoryBuffer.Resize(nSize := requiredSize*SIZEOF(BYTE), bPreserve:=TRUE, bReset:=TRUE);
  _fifo.pBuffer := _dynamicMemoryBuffer.pBuffer;
  _fifo.cbBuffer := requiredSize;
END_IF
END_METHOD

END_FUNCTION_BLOCK
